// TIA Portal project "sayicilarin_zaman_rolesi_ola_kull" (V18)

(* hardware
DEVICE "S7-1200 station_1"  S7-1200 Station
   slot 0: "Rack_0"  S7-1200 Rack  Rack  V1.0
   slot 1: "PLC_1"  CPU 1214C AC/DC/Rly  6ES7 214-1BG40-0XB0  V4.6
*)

// ===== PLC "PLC_1"  CPU 1214C AC/DC/Rly =====

VAR_GLOBAL   // PLC tag table "Default tag table"
   "System_Byte" AT %MB20 : Byte;
   "FirstScan" AT %M20.0 : Bool;
   "DiagStatusUpdate" AT %M20.1 : Bool;
   "AlwaysTRUE" AT %M20.2 : Bool;
   "AlwaysFALSE" AT %M20.3 : Bool;
   "Clock_Byte" AT %MB21 : Byte;
   "Clock_10Hz" AT %M21.0 : Bool;
   "Clock_5Hz" AT %M21.1 : Bool;
   "Clock_2.5Hz" AT %M21.2 : Bool;
   "Clock_2Hz" AT %M21.3 : Bool;
   "Clock_1.25Hz" AT %M21.4 : Bool;
   "Clock_1Hz" AT %M21.5 : Bool;
   "Clock_0.625Hz" AT %M21.6 : Bool;
   "Clock_0.5Hz" AT %M21.7 : Bool;
   "Tag_1" AT %M0.0 : Bool;
   "Tag_2" AT %Q0.0 : Bool;
   "Tag_3" AT %I0.0 : Bool;
   "Tag_4" AT %M100.0 : Bool;
   "Tag_5" AT %I0.1 : Bool;
   "Tag_6" AT %M100.1 : Bool;
   "Tag_7" AT %M100.2 : Bool;
   "Tag_8" AT %M0.1 : Bool;
   "Tag_9" AT %M100.4 : Bool;
   "Tag_10" AT %M100.6 : Bool;
END_VAR

// folder: System blocks/Program resources

DATA_BLOCK "IEC_Counter_0_DB"   // DB1
{ S7_Optimized_Access := 'TRUE' }
AUTHOR : Simatic
FAMILY : IEC
NAME : CNTR
VERSION : 1.0
// stored: InstanceOfName IEC_COUNTER
"IEC_COUNTER"
BEGIN
END_DATA_BLOCK

DATA_BLOCK "C1"   // DB2
{ S7_Optimized_Access := 'TRUE' }
AUTHOR : Simatic
FAMILY : IEC
NAME : CNTR
VERSION : 1.0
// stored: InstanceOfName IEC_COUNTER
"IEC_COUNTER"
BEGIN
END_DATA_BLOCK

// folder: (top level)

ORGANIZATION_BLOCK "Main"   // OB1, LAD, ProgramCycle
TITLE = "Main Program Sweep (Cycle)"
{ S7_Optimized_Access := 'TRUE' }
VERSION : 0.1
   VAR_INPUT
      Initial_Call : Bool;   // Initial call of this OB
      Remanence : Bool;   // =True, if remanent data are available
   END_VAR
   VAR_TEMP   // added for the SCL form of the ladder/FBD networks
      _w1 : Bool;
      _w2 : Bool;
   END_VAR
BEGIN

REGION Network 1
   // Bir motor, start butonuna basıldığında 10sn çalışıp duracak. 5 sn bekledikten sonra yeniden kendiliğinden çalışacak. 10 sn çalışıp yeniden duracaktır. Periyodik çalışma, stop butonuna basılıncaya kadar devam edecektir
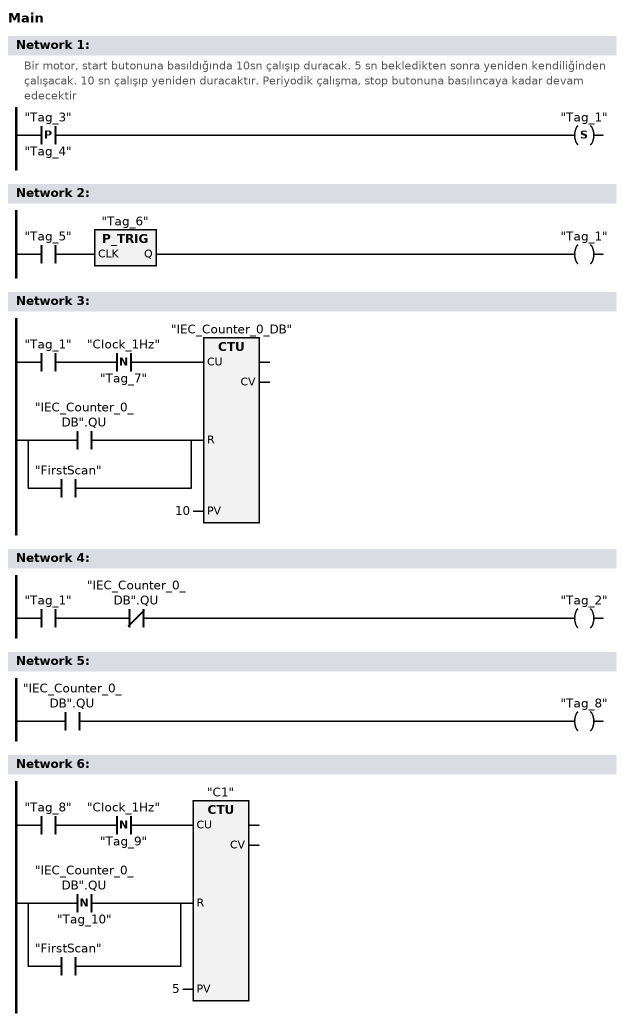
   RUNG wire#powerrail
      P_Contact(operand := "Tag_3", bit := "Tag_4")
      S_Coil( "Tag_1" )
   END_RUNG
   // the same network as SCL:
   #_w1 := "Tag_3" AND NOT "Tag_4";   // rising edge of "Tag_3"
   "Tag_4" := "Tag_3";
   IF #_w1 THEN "Tag_1" := TRUE; END_IF;
END_REGION

REGION Network 2
   RUNG wire#powerrail
      Contact( "Tag_5" )
      P_Trig( "Tag_6" )
      Coil( "Tag_1" )
   END_RUNG
   // the same network as SCL:
   #_w1 := "Tag_5" AND NOT "Tag_6";   // rising edge
   "Tag_6" := "Tag_5";
   "Tag_1" := #_w1;
END_REGION

REGION Network 3
   #_w1 := "Tag_1" AND NOT "Clock_1Hz" AND "Tag_7";   // falling edge of "Clock_1Hz"
   "Tag_7" := "Clock_1Hz";
   "IEC_Counter_0_DB".CTU(CU := #_w1, R := "IEC_Counter_0_DB".QU OR "FirstScan", PV := 10);
END_REGION

REGION Network 4
   RUNG wire#powerrail
      Contact( "Tag_1" )
      I_Contact( "IEC_Counter_0_DB".QU )
      Coil( "Tag_2" )
   END_RUNG
   // the same network as SCL:
   "Tag_2" := "Tag_1" AND NOT "IEC_Counter_0_DB".QU;
END_REGION

REGION Network 5
   RUNG wire#powerrail
      Contact( "IEC_Counter_0_DB".QU )
      Coil( "Tag_8" )
   END_RUNG
   // the same network as SCL:
   "Tag_8" := "IEC_Counter_0_DB".QU;
END_REGION

REGION Network 6
   #_w1 := "Tag_8" AND NOT "Clock_1Hz" AND "Tag_9";   // falling edge of "Clock_1Hz"
   "Tag_9" := "Clock_1Hz";
   #_w2 := NOT "IEC_Counter_0_DB".QU AND "Tag_10";   // falling edge of "IEC_Counter_0_DB".QU
   "Tag_10" := "IEC_Counter_0_DB".QU;
   "C1".CTU(CU := #_w1, R := #_w2 OR "FirstScan", PV := 5);
END_REGION
END_ORGANIZATION_BLOCK